(* IEC 61131-3 sources: FIOWrap/src/Ar/FIOWrap, 8 files *)

(* ---- FIOWrap.typ ---- *)
(*
 * File: FIOWrap.typ
 * Copyright (c) 2023 Loupe
 * https://loupe.team
 *
 * This file is part of FIOWrap, licensed under the MIT License.
 *
 ********************************************************************
 * Data types of library FIOWrap
 ********************************************************************)

TYPE
	FIOWRAP_ERR_enum :
		(
		FIOWRAP_ERR_INVALIDOP := 50000,
		FIOWRAP_ERR_INVALIDFILTER,
		FIOWRAP_ERR_INVALIDDIR,
		FIOWRAP_ERR_MAXFILESIZE
		);
	FIOWRAP_OP_enum :
		(
		FIOWRAP_OP_INVALID := 0,
		FIOWRAP_OP_OPEN,
		FIOWRAP_OP_SAVEAS,
		FIOWRAP_OP_APPEND,
		FIOWRAP_OP_APPEND_NEW,
		FIOWRAP_OP_SCAN,
		FIOWRAP_OP_DELETE,
		FIOWRAP_OP_DELETE_ALL,
		FIOWRAP_OP_ERROR
		);
	FIOWRAP_ST_enum :
		(
		FIOWRAP_ST_WAIT := 0, (*0*)
		FIOWRAP_ST_OPEN, (*1*)
		FIOWRAP_ST_CREATE, (*2*)
		FIOWRAP_ST_WRITE_HEADER, (*3*)
		FIOWRAP_ST_READ, (*4*)
		FIOWRAP_ST_WRITE, (*5*)
		FIOWRAP_ST_CLOSE, (*6*)
		FIOWRAP_ST_DELETE, (*7*)
		FIOWRAP_ST_DELETE_FILE, (*8*)
		FIOWRAP_ST_DELETE_DIR, (*9*)
		FIOWRAP_ST_RENAME, (*10*)
		FIOWRAP_ST_INFO, (*11*)
		FIOWRAP_ST_ERROR := 999, (*999*)
		FIOWRAP_ST_
		);
	FIOWrap_Int_FUB_typ : 	STRUCT
		Open : FileOpen;
		Create : FileCreate;
		Read : FileRead;
		Write : FileWrite;
		Close : FileClose;
		Delete : FileDelete;
		Rename : FileRename;
		GetTime : DTGetTime;
		Info : FileInfo;
	END_STRUCT;
	FIOWrap_Internal_typ : 	STRUCT
		FileID : UDINT; (*File Ident for reading and writing*)
		FileLen : UDINT; (*Length of the current file for appending*)
		FileCreated : BOOL; (*Error happened after opening file.  Need to close and then go to error state.*)
		ErrorClose : BOOL; (*Error happened after opening file.  Need to close and then go to error state.*)
		CurrOperation : DINT;
		State : DINT;
		Timestamp : STRING[30];
		newFileName : STRING[FIOWRAP_STRLEN_NAME];
		Name : STRING[FIOWRAP_STRLEN_NAME];
		Extension : STRING[FIOWRAP_STRLEN_NAME];
		FUB : FIOWrap_Int_FUB_typ;
		CMD : FIOWrap_IN_CMD_typ;
		DTStruct : DTStructure;
		TempStr : STRING[FIOWRAP_STRLEN_NAME];
		FileInfo : fiFILE_INFO;
		headerLen : UDINT;
	END_STRUCT;
	FIOWrap_OUT_STAT_typ : 	STRUCT
		Busy : BOOL;
		Done : BOOL;
		Error : BOOL;
		ErrorID : UINT;
		ErrorString : STRING[FIOWRAP_STRLEN_ERROR];
		ErrorLevel : USINT;
		ReadyForCMD : BOOL;
		NewFile : BOOL; (*Length of the current file for appending*)
		FileLen : UDINT; (*Length of the current file for appending*)
	END_STRUCT;
	FIOWrap_OUT_typ : 	STRUCT
		STAT : FIOWrap_OUT_STAT_typ;
	END_STRUCT;
	FIOWrap_IN_PAR_typ : 	STRUCT
		FileDevice : STRING[FIOWRAP_STRLEN_NAME]; (*File device name*)
		FileName : STRING[FIOWRAP_STRLEN_NAME]; (*File name (with extension)*)
		Suffix : STRING[FIOWRAP_STRLEN_NAME]; (*File name (with extension)*)
		pData : UDINT; (*Address of the data to be read or written*)
		len : UDINT; (*Length of the data to be read or written*)
		offset : UDINT; (*Offset within the file to read/write from/to.*)
		MaxFileSize : UDINT; (*Maximum file size (only evaluated when appending to a file)*)
		MultiFile : BOOL; (*Allow multiple files to be created. When true, AppendToFile will not issue an error if the MaxFileSize would be exceeded. Instead, a new file is created with the name FileName. The original file is renamed to include the FileName and the Suffix.*)
		pHeader : UDINT; (*Address of data to be added to the top of new files*)
		headerLen : UDINT; (*Length or size of header in bytes*)
	END_STRUCT;
	FIOWrap_IN_CMD_typ : 	STRUCT
		Open : BOOL; (*Open a file and read its contents*)
		SaveAs : BOOL; (*Save data to a file*)
		AppendToFile : BOOL; (*Append data to the end of a file*)
		Delete : BOOL;
		AcknowledgeError : BOOL;
	END_STRUCT;
	FIOWrap_IN_typ : 	STRUCT
		CMD : FIOWrap_IN_CMD_typ;
		PAR : FIOWrap_IN_PAR_typ;
	END_STRUCT;
	FIOWrap_typ : 	STRUCT
		IN : FIOWrap_IN_typ;
		OUT : FIOWrap_OUT_typ;
		Internal : FIOWrap_Internal_typ;
	END_STRUCT;
	FIOManage_Int_FUB_typ : 	STRUCT
		DirOpen : DirOpen;
		DirClose : DirClose;
		DirRead : DirReadEx;
		DeleteDir : DirDeleteEx;
		Delete : FileDelete;
	END_STRUCT;
	FIOManage_Internal_typ : 	STRUCT
		DirID : UDINT; (*File Ident for reading and writing*)
		NumDirs : UDINT; (*Length of the current file for appending*)
		NumItems : UDINT; (*Length of the current file for appending*)
		CurrOperation : FIOWRAP_OP_enum;
		ErrorClose : BOOL; (*Error happened after opening file.  Need to close and then go to error state.*)
		State : DINT;
		index : USINT;
		FilterName : STRING[FIOWRAP_STRLEN_NAME];
		ItemName : STRING[FIOWRAP_STRLEN_NAME];
		FileExtension : STRING[FIOWRAP_STRLEN_NAME];
		Name : STRING[FIOWRAP_STRLEN_NAME];
		Extension : STRING[FIOWRAP_STRLEN_NAME];
		NumItemsDelete : DINT;
		ItemInfo : fiDIR_READ_EX_DATA;
		ItemInfoCache : ARRAY[0..FIOWRAP_MAI_DELETE]OF fiDIR_READ_EX_DATA;
		NewestIndex : USINT;
		OldestIndex : USINT;
		FUB : FIOManage_Int_FUB_typ;
		CMD : FIOManage_IN_CMD_typ;
	END_STRUCT;
	FIOManage_OUT_STAT_typ : 	STRUCT
		Busy : BOOL;
		Done : BOOL;
		Error : BOOL;
		ErrorID : UINT;
		ErrorString : STRING[FIOWRAP_STRLEN_ERROR];
		ErrorLevel : USINT;
		ReadyForCMD : BOOL;
	END_STRUCT;
	FIOManage_OUT_typ : 	STRUCT
		STAT : FIOManage_OUT_STAT_typ;
	END_STRUCT;
	FIOManage_IN_PAR_typ : 	STRUCT
		FileDevice : STRING[FIOWRAP_STRLEN_NAME]; (*File device name*)
		Directory : STRING[FIOWRAP_STRLEN_NAME]; (*Directory to navigate to*)
		ItemName : STRING[FIOWRAP_STRLEN_NAME]; (*Address of the data to be read or written*)
		MaxNumItems : UDINT; (*Maximum file size (only evaluated when appending to a file)*)
		Mode : USINT; (*Maximum file size (only evaluated when appending to a file)*)
	END_STRUCT;
	FIOManage_IN_CMD_typ : 	STRUCT
		Scan : BOOL;
		DeleteAll : BOOL;
		AcknowledgeError : BOOL;
	END_STRUCT;
	FIOManage_IN_typ : 	STRUCT
		CMD : FIOManage_IN_CMD_typ;
		PAR : FIOManage_IN_PAR_typ;
	END_STRUCT;
	FIOManage_typ : 	STRUCT
		IN : FIOManage_IN_typ;
		OUT : FIOManage_OUT_typ;
		Internal : FIOManage_Internal_typ;
	END_STRUCT;
END_TYPE

(* ---- FIOManageFn_Cyclic.st ---- *)
(*
 * File: FIOManageFn_Cyclic.st
 * Copyright (c) 2023 Loupe
 * https://loupe.team
 *
 * This file is part of FIOWrap, licensed under the MIT License.
 *
  ********************************************************************
 * Implementation of library FIOWrap
 ********************************************************************)

(********************************************************************)
(* This function manages multiple files for logs					*)
(********************************************************************)

(* Resetting internal CMDs				DONE and NOT TESTED *)

(* Main State machine					DONE NOT TESTED *)

	(* ST_WAIT							DONE NOT TESTED *)
		(* Wait for new CMDs			DONE and TESTED *)
			(* Scan						DONE and TESTED  *)
				(* Set CurrOperation	DONE and TESTED  *)
				(* Busy, Done			DONE and TESTED  *)
				(* Change state			DONE and TESTED  *)
			(* DeleteAll				DONE and NOT TESTED  *)
				(* Set CurrOperation	DONE and TESTED  *)
				(* Busy, Done			DONE and TESTED  *)
				(* Change state			DONE and TESTED  *)
		(* Reset Done					DONE and TESTED  *)

	(* ST_OPEN							DONE and NOT TESTED  *)
		(* FUB inputs					DONE and TESTED  *)
		(* Status checking				DONE and TESTED  *)
			(* Done						DONE and TESTED  *)
			(* No error					DONE and TESTED  *)
				(* Open					DONE and TESTED  *)
			(* Other error				DONE and NOT TESTED  *)

	(* ST_READ							DONE and NOT TESTED  *)
		(* FUB inputs					DONE and NOT TESTED  *)
		(* Status checking				DONE and NOT TESTED  *)
			(* Done						DONE and TESTED  *)
			(* No error					DONE and TESTED  *)
			(* Error					DONE and TESTED  *)

	(* ST_CLOSE							DONE and NOT TESTED  *)
		(* FUB inputs					DONE and NOT TESTED  *)
		(* Status checking				DONE and NOT TESTED  *)
			(* Done						DONE and TESTED  *)
			(* No error					DONE and TESTED  *)
				(* ErrorClose			DONE and NOT TESTED  *)
			(* Error					DONE will not be tested *)

	(* ST_DELETE						DONE and NOT TESTED  *)
		(* FUB inputs					DONE and NOT TESTED  *)
		(* Status checking				DONE and NOT TESTED  *)
			(* Done						DONE and TESTED  *)
			(* No error					DONE and TESTED  *)
			(* File not found			DONE and NOT TESTED  *)
			(* Other error				DONE and NOT TESTED  *)

	(* ST_ERROR							DONE and TESTED  *)
		(* Disable FUBs					DONE and TESTED  *)
		(* AcknowledgeError CMD			DONE and TESTED  *)

(* Busy, Done, Error					DONE and TESTED  *)

FUNCTION FIOManageFn_Cyclic

(************************************************************************)
(* Set return value to get rid of compiler warning 						*)
(************************************************************************)

FIOManageFn_Cyclic:=	FALSE;

(************************************************************************)
(* Reset internal CMDs													*)
(************************************************************************)

IF( NOT(t.IN.CMD.Scan) )THEN

	t.Internal.CMD.Scan:=	0;

END_IF

IF( NOT(t.IN.CMD.DeleteAll) )THEN

	t.Internal.CMD.DeleteAll:=	0;

END_IF

(************************************************************************)
(* Main state machine													*)
(************************************************************************)

	CASE t.Internal.State OF

		FIOWRAP_ST_WAIT:

			(* If all CMDs are cleared, then clear Done status *)

			IF( 	NOT(t.IN.CMD.Scan)
				AND	NOT(t.IN.CMD.DeleteAll)
				)THEN

				t.OUT.STAT.Done:=	0;

			END_IF

			(* Set CurrOperation to INVALID. It will be set below on leaving the state *)

			t.Internal.CurrOperation:=	FIOWRAP_OP_INVALID;

			(* Wait for new commands *)

			IF( t.IN.CMD.Scan AND NOT(t.Internal.CMD.Scan) )THEN

				t.Internal.CMD.Scan:=	1;

				t.OUT.STAT.Busy:=	1;
				t.OUT.STAT.Done:=	0;

				t.Internal.State:=			FIOWRAP_ST_OPEN;
				t.Internal.CurrOperation:=	FIOWRAP_OP_SCAN;

				// Modify filter based off of input itemName
				IF(t.IN.PAR.ItemName = '') THEN
					// Set error for filter input
					fiomSetError( DINT_TO_UINT(FIOWRAP_ERR_INVALIDFILTER), t );
				ELSIF (t.IN.PAR.ItemName = '*') THEN
					t.Internal.FilterName := '';
				ELSE
					t.Internal.FilterName := t.IN.PAR.ItemName;
				END_IF

			ELSIF( t.IN.CMD.DeleteAll AND NOT(t.Internal.CMD.DeleteAll) )THEN

				// TODO: Delete All should not open file more than once

				t.Internal.CMD.DeleteAll:=	1;

				t.OUT.STAT.Busy:=	1;
				t.OUT.STAT.Done:=	0;

				t.Internal.State:=			FIOWRAP_ST_OPEN;
				t.Internal.CurrOperation:=	FIOWRAP_OP_DELETE_ALL;

			END_IF

		FIOWRAP_ST_OPEN:

			(* Open Dir *)

			t.Internal.FUB.DirOpen.enable:=	1;
			t.Internal.FUB.DirOpen.pDevice:=	ADR(t.IN.PAR.FileDevice);
			IF( brsstrlen(ADR(t.IN.PAR.Directory)) = 0 )THEN
				t.Internal.FUB.DirOpen.pName:= 0;
				// Scanning/deleting is not allowed while in a root directory
				// TODO: figure out how to throw an error because figuring out if you are in a root directory is difficult
			ELSE
				t.Internal.FUB.DirOpen.pName:=		ADR(t.IN.PAR.Directory);
			END_IF

			(* Check status *)

			IF( t.Internal.FUB.DirOpen.status < FIOWRAP_STAT_DISABLED ) THEN

				(* Turn off FUB *)

				t.Internal.FUB.DirOpen.enable:=	0;

				IF( t.Internal.FUB.DirOpen.status = FIOWRAP_STAT_OK ) THEN

				(* All good
					Get Ident, go to appropriate state *)

					t.Internal.DirID:=		t.Internal.FUB.DirOpen.ident;

					IF( t.Internal.CurrOperation = FIOWRAP_OP_DELETE
						OR t.Internal.CurrOperation = FIOWRAP_OP_DELETE_ALL
						OR t.Internal.CurrOperation = FIOWRAP_OP_SCAN)THEN

						t.Internal.State:= FIOWRAP_ST_READ;

					ELSE

						fiomSetError( DINT_TO_UINT(FIOWRAP_ERR_INVALIDOP), t );

					END_IF

				ELSE

					(* Other error *)

					fiomSetError( t.Internal.FUB.DirOpen.status, t );

				END_IF (* If error *)

		END_IF (* If done *)

		FIOWRAP_ST_READ:

			(* Check status *)

			IF( t.Internal.FUB.DirRead.status < FIOWRAP_STAT_DISABLED )THEN

				(* Turn off FUB *)

				t.Internal.FUB.DirRead.enable:= 0;

				IF ( t.Internal.FUB.DirRead.status = FIOWRAP_STAT_OK ) THEN

					(* Turn on FUB *)
					t.Internal.FUB.DirRead.enable:= 1;

					// Check mode and file type before adding to the cache
					IF( (t.IN.PAR.Mode = fiFILE AND t.Internal.ItemInfo.Mode = fiFILE)
						OR (t.IN.PAR.Mode = fiDIRECTORY AND t.Internal.ItemInfo.Mode = fiDIRECTORY)
						OR (t.IN.PAR.Mode = fiBOTH) )THEN

						(* Get File Names and Extensions *)
						SplitFileName(ADR(t.Internal.FilterName),ADR(t.Internal.Name), ADR(t.Internal.Extension));
						SplitFileName(ADR(t.Internal.ItemInfo.Filename),0,ADR(t.Internal.FileExtension));
						brsmemcpy(ADR(t.Internal.ItemName),ADR(t.Internal.ItemInfo.Filename),brsstrlen(ADR(t.Internal.Name)));

						// Check to see if the file/directory name and extension (if specified) match and that the directory is not '.' or '..'
						IF( (brsstrcmp(ADR(t.Internal.ItemName),ADR(t.Internal.Name)) = 0)
							AND ((brsstrcmp(ADR(t.Internal.FileExtension),ADR(t.Internal.Extension)) = 0) OR (brsstrcmp(ADR(t.Internal.Extension),ADR('')) = 0))
							AND NOT ((brsstrcmp(ADR(t.Internal.ItemInfo.Filename),ADR('.')) = 0) OR (brsstrcmp(ADR(t.Internal.ItemInfo.Filename),ADR('..')) = 0) ))THEN
							// increment number of files
							t.Internal.NumItems:= t.Internal.NumItems+1;

							// All indices in the cache are set to very large dates initially
							IF( t.Internal.ItemInfoCache[t.Internal.NewestIndex].Date > t.Internal.ItemInfo.Date )THEN

								(* Record Older file info *)
								brsmemcpy(ADR(t.Internal.ItemInfoCache[t.Internal.NewestIndex]),ADR(t.Internal.ItemInfo),SIZEOF(t.Internal.ItemInfo));

								(* Find Oldest / Newest file *)
								FOR t.Internal.index := 0 TO FIOWRAP_MAI_DELETE DO
									IF t.Internal.ItemInfoCache[t.Internal.OldestIndex].Date > t.Internal.ItemInfoCache[t.Internal.index].Date THEN
										t.Internal.OldestIndex := t.Internal.index;
									END_IF
									IF  t.Internal.ItemInfoCache[t.Internal.NewestIndex].Date < t.Internal.ItemInfoCache[t.Internal.index].Date THEN
										t.Internal.NewestIndex := t.Internal.index;
									END_IF
								END_FOR;
							END_IF

							// Start deleting files if you have the max number of files you can delete in one read.
							IF( t.Internal.NumItems >=  FIOWRAP_NUM_DELETE
								AND t.Internal.CurrOperation = FIOWRAP_OP_DELETE_ALL )THEN

								t.Internal.FUB.DirRead.enable:= 0;

								t.Internal.NumItemsDelete:= FIOWRAP_NUM_DELETE;

								(* Delete files *)

								t.Internal.State := FIOWRAP_ST_DELETE;

							END_IF

						END_IF

					END_IF

				ELSIF ( t.Internal.FUB.DirRead.status = fiERR_NO_MORE_ENTRIES ) THEN

					IF t.Internal.CurrOperation = FIOWRAP_OP_DELETE_ALL THEN

						(* Delete Files *)

						t.Internal.NumItemsDelete:= MIN(t.Internal.NumItems, FIOWRAP_NUM_DELETE);

						IF t.Internal.NumItemsDelete > 0 THEN
							t.Internal.CurrOperation := FIOWRAP_OP_DELETE;
						ELSE
							t.Internal.CurrOperation := FIOWRAP_OP_SCAN; //TODO: Change this to valid op
						END_IF

					ELSIF t.Internal.NumItems > t.IN.PAR.MaxNumItems THEN

						(* Delete Files *)

						t.Internal.NumItemsDelete:= MIN(t.Internal.NumItems - t.IN.PAR.MaxNumItems, FIOWRAP_NUM_DELETE);

						t.Internal.CurrOperation := FIOWRAP_OP_DELETE;

					END_IF

					IF( t.Internal.CurrOperation = FIOWRAP_OP_DELETE
						OR t.Internal.CurrOperation = FIOWRAP_OP_DELETE_ALL
						OR t.Internal.CurrOperation = FIOWRAP_OP_SCAN )THEN

						(* Close Dir *)

						t.Internal.State := FIOWRAP_ST_CLOSE;

					ELSE

						fiomSetError( DINT_TO_UINT(FIOWRAP_ERR_INVALIDOP), t );

					END_IF

				ELSE

					(* Error *)

					t.Internal.ErrorClose:= 1;

					IF( t.Internal.FUB.DirRead.status = 20799 )THEN

						//If the sysError ID = 65535 then we are in a root directory and can't do a read
						t.OUT.STAT.ErrorID := FileIoGetSysError();
						IF (t.OUT.STAT.ErrorID = 65535) THEN
							fiomSetError( DINT_TO_UINT(FIOWRAP_ERR_INVALIDDIR), t );
						ELSE
							fiomSetError( t.OUT.STAT.ErrorID, t );
						END_IF

					ELSE

						fiomSetError( t.Internal.FUB.DirRead.status, t );

					END_IF

					t.Internal.State:= FIOWRAP_ST_CLOSE;

				END_IF

			ELSIF( t.Internal.FUB.DirRead.status = FIOWRAP_STAT_DISABLED )THEN

				(* Enable FUB *)
				t.Internal.FUB.DirRead.enable 	:= 1;
				t.Internal.FUB.DirRead.ident	:= t.Internal.DirID;
				t.Internal.FUB.DirRead.pData	:= ADR(t.Internal.ItemInfo);
				t.Internal.FUB.DirRead.data_len	:= SIZEOF(t.Internal.ItemInfo);

				t.Internal.NumItems := 0;
				t.Internal.NumItemsDelete:= 0;
				t.Internal.OldestIndex := 0;
				t.Internal.NewestIndex := 0;
				brsmemset(ADR(t.Internal.ItemName), 0, SIZEOF(t.Internal.ItemName));

				brsmemset(ADR(t.Internal.ItemInfoCache), 0, SIZEOF(t.Internal.ItemInfoCache));
				FOR t.Internal.index := 0 TO FIOWRAP_MAI_DELETE DO
					t.Internal.ItemInfoCache[t.Internal.index].Date := DT#2106-02-06-06:28:15; // Can this be a hex value instead?
				END_FOR

			END_IF

		FIOWRAP_ST_CLOSE:

			(* Close file *)

			t.Internal.FUB.DirClose.enable:=	1;
			t.Internal.FUB.DirClose.ident:=	t.Internal.DirID;

			(* Check status *)

			IF( t.Internal.FUB.DirClose.status < FIOWRAP_STAT_DISABLED ) THEN

				(* Turn off FUB *)

				t.Internal.FUB.DirClose.enable:=	0;

				IF( t.Internal.FUB.DirClose.status = FIOWRAP_STAT_OK ) THEN

					IF( t.Internal.ErrorClose ) THEN

						(* If error, go to error state *)

						t.Internal.State:=	FIOWRAP_ST_ERROR;

						t.Internal.ErrorClose:= 0;

					ELSIF( (t.Internal.CurrOperation = FIOWRAP_OP_DELETE
						OR t.Internal.CurrOperation = FIOWRAP_OP_DELETE_ALL)
						AND t.Internal.NumItemsDelete > 0) THEN

						t.Internal.State:=	FIOWRAP_ST_DELETE;

					ELSE

						(* otherwise, done, set status and go to wait state *)

						t.OUT.STAT.Busy:=	0;
						t.OUT.STAT.Done:=	1;

						t.Internal.State:=	FIOWRAP_ST_WAIT;

					END_IF (* If ErrorClose *)

				ELSE

					(* Error *)

					fiomSetError( t.Internal.FUB.DirClose.status, t );

				END_IF (* If error *)

		END_IF (*If done *)

		FIOWRAP_ST_DELETE:

			IF( t.Internal.NumItemsDelete > 0 )THEN

				(* Generate file name *)

				brsmemcpy(ADR(t.Internal.ItemName),ADR(t.Internal.ItemInfoCache[t.Internal.OldestIndex].Filename),SIZEOF(t.Internal.ItemName));
				t.Internal.ItemName := CONCAT(CONCAT(t.IN.PAR.Directory, '/'), t.Internal.ItemName);

				// Check file type and go to appropriate state
				IF(t.Internal.ItemInfoCache[t.Internal.OldestIndex].Mode = fiFILE) THEN
					t.Internal.State := FIOWRAP_ST_DELETE_FILE;
				ELSE
					t.Internal.State := FIOWRAP_ST_DELETE_DIR;
				END_IF

				(* Remove Old file from list *)

				t.Internal.ItemInfoCache[t.Internal.OldestIndex].Date := DT#2106-02-06-06:28:15; // Can this be a hex value instead?

				(* Find new oldest / newest file *)

				FOR t.Internal.index := 0 TO FIOWRAP_MAI_DELETE DO
					IF t.Internal.ItemInfoCache[t.Internal.OldestIndex].Date > t.Internal.ItemInfoCache[t.Internal.index].Date THEN
						t.Internal.OldestIndex := t.Internal.index;
					END_IF
					IF  t.Internal.ItemInfoCache[t.Internal.NewestIndex].Date < t.Internal.ItemInfoCache[t.Internal.index].Date THEN
						t.Internal.NewestIndex := t.Internal.index;
					END_IF
				END_FOR;

			ELSIF( t.Internal.NumItemsDelete <= 0 )THEN

				IF( t.Internal.CurrOperation = FIOWRAP_OP_DELETE_ALL )THEN

					(* Go to Read *)
					// Find more files to delete
					t.Internal.State:= FIOWRAP_ST_OPEN;

				ELSIF( t.Internal.CurrOperation = FIOWRAP_OP_DELETE )THEN

					(* Done, set status and go to wait state *)
					t.OUT.STAT.Busy:=	0;
					t.OUT.STAT.Done:=	1;

					t.Internal.State:=	FIOWRAP_ST_WAIT;

				ELSE
					// Set the error
					fiomSetError( DINT_TO_UINT(FIOWRAP_ERR_INVALIDOP), t );

				END_IF

			END_IF

		FIOWRAP_ST_DELETE_FILE:
			(* Enable FUB *)
			IF (NOT t.Internal.FUB.Delete.enable) THEN
				t.Internal.FUB.Delete.enable := 1;
				t.Internal.FUB.Delete.pDevice := ADR(t.IN.PAR.FileDevice);
				t.Internal.FUB.Delete.pName := ADR(t.Internal.ItemName);
			END_IF

			(*Delete File*)
			IF( t.Internal.FUB.Delete.status < FIOWRAP_STAT_DISABLED )THEN

				(* Turn off FUB *)
				t.Internal.FUB.Delete.enable:= 0;

				IF( t.Internal.FUB.Delete.status = FIOWRAP_STAT_OK )THEN

					t.Internal.NumItems := t.Internal.NumItems - 1;
					t.Internal.NumItemsDelete := t.Internal.NumItemsDelete - 1;

					// Return to delete state
					t.Internal.State := FIOWRAP_ST_DELETE;

				ELSE

					(* error *)

					//TODO: Handle file not found error

					fiomSetError( t.Internal.FUB.Delete.status, t );

				END_IF
			END_IF

		FIOWRAP_ST_DELETE_DIR:
			(* Enable FUB *)
			IF (NOT t.Internal.FUB.DeleteDir.enable) THEN
				t.Internal.FUB.DeleteDir.enable := 1;
				t.Internal.FUB.DeleteDir.pDevice := ADR(t.IN.PAR.FileDevice);
				t.Internal.FUB.DeleteDir.pName := ADR(t.Internal.ItemName);
			END_IF

			(*Delete File*)

			IF( t.Internal.FUB.DeleteDir.status < FIOWRAP_STAT_DISABLED )THEN

				(* Turn off FUB *)

				t.Internal.FUB.DeleteDir.enable:= 0;

				IF( t.Internal.FUB.DeleteDir.status = FIOWRAP_STAT_OK )THEN

					t.Internal.NumItems := t.Internal.NumItems - 1;
					t.Internal.NumItemsDelete := t.Internal.NumItemsDelete - 1;

					// Return to delete state
					t.Internal.State := FIOWRAP_ST_DELETE;

				ELSE

					(* error *)

					//TODO: Handle file not found error

					fiomSetError( t.Internal.FUB.DeleteDir.status, t );

				END_IF
			END_IF

		FIOWRAP_ST_ERROR:

			(* Turn off all FUBs, just in case *)

			t.Internal.FUB.DirOpen.enable:=	0;
			t.Internal.FUB.DirRead.enable:=	0;
			t.Internal.FUB.DirClose.enable:=	0;
			t.Internal.FUB.Delete.enable:=	0;

			IF( t.IN.CMD.AcknowledgeError )THEN

				t.OUT.STAT.Error:=			0;
				t.OUT.STAT.ErrorID:=		0;
				t.OUT.STAT.ErrorString:=	'';
				t.OUT.STAT.ErrorLevel:=		0;
				t.Internal.State:=			FIOWRAP_ST_WAIT;

			END_IF

	END_CASE

	(* Reset AcknowledgeError CMD *)

	t.IN.CMD.AcknowledgeError:=	0;

	(****************************************)
	(* Call FUBs							*)
	(****************************************)

	t.Internal.FUB.DirOpen();
	t.Internal.FUB.DirRead();
	t.Internal.FUB.DirClose();
	t.Internal.FUB.Delete();
	t.Internal.FUB.DeleteDir();

(****************************************)
(* Set ReadyForCMD						*)
(****************************************)

t.OUT.STAT.ReadyForCMD:=		NOT(t.OUT.STAT.Busy)
							AND NOT(t.OUT.STAT.Done)
							AND	NOT(t.OUT.STAT.Error);

END_FUNCTION

(* ---- fiomSetError.st ---- *)
(*
 * File: fiomSetError.st
 * Copyright (c) 2023 Loupe
 * https://loupe.team
 *
 * This file is part of FIOWrap, licensed under the MIT License.
 *
  ********************************************************************
 * Implementation of library FIOWrap
 ********************************************************************)

(********************************************************************)
(* Set error status on FIOWrap 										*)
(********************************************************************)

(* Reset Busy, Done			DONE and TESTED DFB 20111222 *)
(* Set Error				DONE and TESTED DFB 20111222 *)
(* Set ErrorID				DONE and TESTED DFB 20111222 *)
(* Set ErrorLevel			DONE and TESTED DFB 20111222 *)
(* Set State				DONE and TESTED DFB 20111222 *)
(* Set ErrorString			DONE and TESTED DFB 20120131 *)

FUNCTION fiomSetError

(****************************************************)
(* Set return value to get rid of compile warning 	*)
(****************************************************)

fiomSetError:=	FALSE;

(************************************************)
(* Set error status								*)
(************************************************)

t.OUT.STAT.Busy:=		0;
t.OUT.STAT.Done:=		0;
t.OUT.STAT.Error:=		1;
t.OUT.STAT.ErrorID:=	ErrorID;
t.OUT.STAT.ErrorLevel:=	3;
t.Internal.State:=		FIOWRAP_ST_ERROR;

(* Set ErrorString *)

CASE ErrorID OF

	0: t.OUT.STAT.ErrorString:=	'';

	fiERR_INVALID_PATH:				t.OUT.STAT.ErrorString:=	'Invalid path.';
	fiERR_DATA_SIZE:				t.OUT.STAT.ErrorString:=	'Data length is too small (DirRead).';
	fiERR_NO_MORE_ENTRIES:			t.OUT.STAT.ErrorString:=	'No more file handles available.';
	fiERR_NOT_SUPPORTED:			t.OUT.STAT.ErrorString:=	'System error.';
	fiERR_INVALID_TYP:				t.OUT.STAT.ErrorString:=	'Invalid type.';
	fiERR_EXIST:					t.OUT.STAT.ErrorString:=	'File already exists.';
	fiERR_ACCESS:					t.OUT.STAT.ErrorString:=	'Access not possible with the desired mode.';
	fiERR_MODE:						t.OUT.STAT.ErrorString:=	'Illegal mode.';
	fiERR_FILE_NOT_FOUND:			t.OUT.STAT.ErrorString:=	'File not found. Check IN.PAR.FileName.';
	fiERR_FILE_DEVICE:				t.OUT.STAT.ErrorString:=	'File device not found. Check IN.PAR.FileDevice.';
	fiERR_SPACE:					t.OUT.STAT.ErrorString:=	'Not enough memory to write file.';
	fiERR_SEEK:						t.OUT.STAT.ErrorString:=	'Invalid file offset.';
	fiERR_FILE:						t.OUT.STAT.ErrorString:=	'File not allowed.';
	fiERR_LESS_VIRTUAL_MEMORY:		t.OUT.STAT.ErrorString:=	'Not enough memory to write file.';
	fiERR_COM_FILE_OPEN:			t.OUT.STAT.ErrorString:=	'System error.';
	fiERR_COM_FILE_CLOSE:			t.OUT.STAT.ErrorString:=	'System error.';
	fiERR_COM_FILE_READ:			t.OUT.STAT.ErrorString:=	'System error.';
	fiERR_COM_FILE_WRITE:			t.OUT.STAT.ErrorString:=	'System error.';
	fiERR_COM_FILE_IOCTL:			t.OUT.STAT.ErrorString:=	'System error.';
	fiERR_DATA:						t.OUT.STAT.ErrorString:=	'Invalid parameter. Check IN.PAR.pData.';
	fiERR_ASYNC_MANAGER:			t.OUT.STAT.ErrorString:=	'System error.';
	fiERR_FILE_NOT_OPENED:			t.OUT.STAT.ErrorString:=	'File not opened.';
	fiERR_INVALID_DIRECTORY:		t.OUT.STAT.ErrorString:=	'Invalid directory. Check IN.PAR.FileDevice and IN.PAR.FileDirectory.';
	fiERR_DIR_NOT_EXIST:			t.OUT.STAT.ErrorString:=	'Directory does not exist. Check IN.PAR.FileDevice and IN.PAR.FileDirectory.';
	fiERR_DIR_NOT_EMPTY:			t.OUT.STAT.ErrorString:=	'Directory is not empty.';
	fiERR_DIR_ALREADY_EXIST:		t.OUT.STAT.ErrorString:=	'Directory already exists.';
	fiERR_DETMEMINFO:				t.OUT.STAT.ErrorString:=	'System error.';
	fiERR_NOT_ENOUGH_FREEMEM:		t.OUT.STAT.ErrorString:=	'Not enough memory to write file.';
	fiERR_DIR_INVALID_HANDLE:		t.OUT.STAT.ErrorString:=	'System error.';
	fiERR_PARAMETER:				t.OUT.STAT.ErrorString:=	'System error.';
	fiERR_DEVICE_ALREADY_EXIST:		t.OUT.STAT.ErrorString:=	'Device already exists.';
	fiERR_DEVICE_INVALID_HANDLE:	t.OUT.STAT.ErrorString:=	'Invalid device handle.';
	fiERR_NETIO_IP_UNEQUAL:			t.OUT.STAT.ErrorString:=	'IP address error. Check hostname.';
	fiERR_INIT:						t.OUT.STAT.ErrorString:=	'System error.';
	fiERR_DEVICE_DRIVER:			t.OUT.STAT.ErrorString:=	'System error.';
	fiERR_DEVICE_MANAGER:			t.OUT.STAT.ErrorString:=	'File device error. Check IN.PAR.FileDevice.';
	fiERR_SYSTEM:					t.OUT.STAT.ErrorString:=	'System error.';

	FIOWRAP_ERR_INVALIDOP:			t.OUT.STAT.ErrorString:=	'Internal error.';
	FIOWRAP_ERR_INVALIDFILTER:		t.OUT.STAT.ErrorString:=	'Input required for IN.PAR.ItemName. Set IN.PAR.ItemName := $'*$' to mamange all files/directories.';
	FIOWRAP_ERR_INVALIDDIR:			t.OUT.STAT.ErrorString:=	'Cannot manage in root directory. Check IN.PAR.FileDevice and IN.PAR.FileDirectory.';
	FIOWRAP_ERR_MAXFILESIZE:		t.OUT.STAT.ErrorString:=	'Error while appending: maximum file size would be exceeded.';

	ELSE	t.OUT.STAT.ErrorString:=	'Unknown error.';

END_CASE

END_FUNCTION

(* ---- fioOpenFile_Init.st ---- *)
(*
 * File: fioOpenFile_Init.st
 * Copyright (c) 2023 Loupe
 * https://loupe.team
 *
 * This file is part of FIOWrap, licensed under the MIT License.
 *
 *)

//-------------------------------------------------------------------
// Open a file in the init subroutine
//-------------------------------------------------------------------

FUNCTION fioOpenFile_Init

	// Open a file - tested
	WHILE (TRUE) DO

		t.IN.CMD.Open := TRUE;

		FIOWrapFn_Cyclic(t);

		IF (t.OUT.STAT.Done OR t.OUT.STAT.Error) THEN
			t.IN.CMD.Open := FALSE;
			FIOWrapFn_Cyclic(t);
			fioOpenFile_Init := t.OUT.STAT.ErrorID;
			RETURN;
		END_IF

	END_WHILE

END_FUNCTION

(* ---- FIOWrap.fun ---- *)
(*
 * File: FIOWrap.fun
 * Copyright (c) 2023 Loupe
 * https://loupe.team
 *
 * This file is part of FIOWrap, licensed under the MIT License.
 *
 ********************************************************************
 * Functions and function blocks of library FIOWrap
 ********************************************************************)

FUNCTION FIOManageFn_Cyclic : BOOL
	VAR_IN_OUT
		t : FIOManage_typ;
	END_VAR
END_FUNCTION

FUNCTION FIOWrapFn_Cyclic : BOOL (*This function manages file reads and writes.*)
	VAR_IN_OUT
		t : FIOWrap_typ; (*FIOWrap Mgr structure*)
	END_VAR
END_FUNCTION

FUNCTION fiowSetError : BOOL (*Set error status on FIOWrap*)
	VAR_INPUT
		ErrorID : UINT;
	END_VAR
	VAR_IN_OUT
		t : FIOWrap_typ;
	END_VAR
END_FUNCTION

FUNCTION fiomSetError : BOOL
	VAR_INPUT
		ErrorID : UINT;
	END_VAR
	VAR_IN_OUT
		t : FIOManage_typ;
	END_VAR
END_FUNCTION

{REDUND_ERROR} FUNCTION fioOpenFile_Init : UINT (*Open a file in the init subroutine*) (*$GROUP=User,$CAT=User,$GROUPICON=User.png,$CATICON=User.png*)
	VAR_IN_OUT
		t : FIOWrap_typ;
	END_VAR
END_FUNCTION

(* ---- fiowSetError.st ---- *)
(*
 * File: fiowSetError.st
 * Copyright (c) 2023 Loupe
 * https://loupe.team
 *
 * This file is part of FIOWrap, licensed under the MIT License.
 *
 ********************************************************************
 * Implementation of library FIOWrap
 ********************************************************************)

(********************************************************************)
(* Set error status on FIOWrap 										*)
(********************************************************************)

(* Reset Busy, Done			DONE and TESTED DFB 20111222 *)
(* Set Error				DONE and TESTED DFB 20111222 *)
(* Set ErrorID				DONE and TESTED DFB 20111222 *)
(* Set ErrorLevel			DONE and TESTED DFB 20111222 *)
(* Set State				DONE and TESTED DFB 20111222 *)
(* Set ErrorString			DONE and TESTED DFB 20120131 *)

FUNCTION fiowSetError

(****************************************************)
(* Set return value to get rid of compile warning 	*)
(****************************************************)

fiowSetError:=	FALSE;

(************************************************)
(* Set error status								*)
(************************************************)

t.OUT.STAT.Busy:=		0;
t.OUT.STAT.Done:=		0;
t.OUT.STAT.Error:=		1;
t.OUT.STAT.ErrorID:=	ErrorID;
t.OUT.STAT.ErrorLevel:=	3;
t.Internal.State:=		FIOWRAP_ST_ERROR;

(* Set ErrorString *)

CASE ErrorID OF

	0: t.OUT.STAT.ErrorString:=	'';

	fiERR_INVALID_PATH:				t.OUT.STAT.ErrorString:=	'Invalid path.';
	fiERR_DATA_SIZE:				t.OUT.STAT.ErrorString:=	'Data length is too small (DirRead).';
	fiERR_NO_MORE_ENTRIES:			t.OUT.STAT.ErrorString:=	'No more file handles available.';
	fiERR_NOT_SUPPORTED:			t.OUT.STAT.ErrorString:=	'System error.';
	fiERR_INVALID_TYP:				t.OUT.STAT.ErrorString:=	'Invalid type.';
	fiERR_EXIST:					t.OUT.STAT.ErrorString:=	'File already exists.';
	fiERR_ACCESS:					t.OUT.STAT.ErrorString:=	'Access not possible with the desired mode.';
	fiERR_MODE:						t.OUT.STAT.ErrorString:=	'Illegal mode.';
	fiERR_FILE_NOT_FOUND:			t.OUT.STAT.ErrorString:=	'File not found. Check IN.PAR.FileName.';
	fiERR_FILE_DEVICE:				t.OUT.STAT.ErrorString:=	'File device not found. Check IN.PAR.FileDevice.';
	fiERR_SPACE:					t.OUT.STAT.ErrorString:=	'Not enough memory to write file.';
	fiERR_SEEK:						t.OUT.STAT.ErrorString:=	'Invalid file offset.';
	fiERR_FILE:						t.OUT.STAT.ErrorString:=	'File not allowed.';
	fiERR_LESS_VIRTUAL_MEMORY:		t.OUT.STAT.ErrorString:=	'Not enough memory to write file.';
	fiERR_COM_FILE_OPEN:			t.OUT.STAT.ErrorString:=	'System error.';
	fiERR_COM_FILE_CLOSE:			t.OUT.STAT.ErrorString:=	'System error.';
	fiERR_COM_FILE_READ:			t.OUT.STAT.ErrorString:=	'System error.';
	fiERR_COM_FILE_WRITE:			t.OUT.STAT.ErrorString:=	'System error.';
	fiERR_COM_FILE_IOCTL:			t.OUT.STAT.ErrorString:=	'System error.';
	fiERR_DATA:						t.OUT.STAT.ErrorString:=	'Invalid parameter. Check IN.PAR.pData.';
	fiERR_ASYNC_MANAGER:			t.OUT.STAT.ErrorString:=	'System error.';
	fiERR_FILE_NOT_OPENED:			t.OUT.STAT.ErrorString:=	'File not opened.';
	fiERR_INVALID_DIRECTORY:		t.OUT.STAT.ErrorString:=	'Invalid directory. Check IN.PAR.FileDevice and IN.PAR.FileName.';
	fiERR_DIR_NOT_EXIST:			t.OUT.STAT.ErrorString:=	'Directory does not exist. Check IN.PAR.FileDevice and IN.PAR.FileName.';
	fiERR_DIR_NOT_EMPTY:			t.OUT.STAT.ErrorString:=	'Directory is not empty.';
	fiERR_DIR_ALREADY_EXIST:		t.OUT.STAT.ErrorString:=	'Directory already exists.';
	fiERR_DETMEMINFO:				t.OUT.STAT.ErrorString:=	'System error.';
	fiERR_NOT_ENOUGH_FREEMEM:		t.OUT.STAT.ErrorString:=	'Not enough memory to write file.';
	fiERR_DIR_INVALID_HANDLE:		t.OUT.STAT.ErrorString:=	'System error.';
	fiERR_PARAMETER:				t.OUT.STAT.ErrorString:=	'System error.';
	fiERR_DEVICE_ALREADY_EXIST:		t.OUT.STAT.ErrorString:=	'Device already exists.';
	fiERR_DEVICE_INVALID_HANDLE:	t.OUT.STAT.ErrorString:=	'Invalid device handle.';
	fiERR_NETIO_IP_UNEQUAL:			t.OUT.STAT.ErrorString:=	'IP address error. Check hostname.';
	fiERR_INIT:						t.OUT.STAT.ErrorString:=	'System error.';
	fiERR_DEVICE_DRIVER:			t.OUT.STAT.ErrorString:=	'System error.';
	fiERR_DEVICE_MANAGER:			t.OUT.STAT.ErrorString:=	'File device error. Check IN.PAR.FileDevice.';
	fiERR_SYSTEM:					t.OUT.STAT.ErrorString:=	'System error.';

	FIOWRAP_ERR_INVALIDOP:			t.OUT.STAT.ErrorString:=	'Internal error.';
	FIOWRAP_ERR_MAXFILESIZE:		t.OUT.STAT.ErrorString:=	'Error while appending: maximum file size would be exceeded.';

	ELSE	t.OUT.STAT.ErrorString:=	'Unknown error.';

END_CASE

END_FUNCTION

(* ---- FIOWrap.var ---- *)
(*
 * File: FIOWrap.var
 * Copyright (c) 2023 Loupe
 * https://loupe.team
 *
 * This file is part of FIOWrap, licensed under the MIT License.
 *
 ********************************************************************
 * Constants of library FIOWrap
 ********************************************************************)
VAR CONSTANT
	FIOWRAP_STRLEN_ERROR : USINT := 120;
	FIOWRAP_NUM_DELETE : USINT := 10;
	FIOWRAP_MAI_DELETE : USINT := FIOWRAP_NUM_DELETE-1;
	FIOWRAP_STRLEN_NAME : UINT := 260;
	FIOWRAP_STAT_OK : UINT := 0;
	FIOWRAP_STAT_DISABLED : UINT := 65534;
END_VAR

(* ---- FIOWrapFn_Cyclic.st ---- *)
(*
 * File: FIOWrapFn_Cyclic.st
 * Copyright (c) 2023 Loupe
 * https://loupe.team
 *
 * This file is part of FIOWrap, licensed under the MIT License.
 *
 ********************************************************************
 * Implementation of library FIOWrap
 ********************************************************************)

(********************************************************************)
(* This function manages simple file reads and writes				*)
(********************************************************************)

(* Resetting internal CMDs				DONE and TESTED DFB 20110602 *)

(* Main State machine					DONE and TESTED DFB 20110602 *)

	(* ST_WAIT							DONE and TESTED DFB 20110602 *)
		(* Wait for new CMDs			DONE and TESTED DFB 20110602 *)
			(* SaveAs					DONE and TESTED DFB 20110602 *)
				(* Set CurrOperation	DONE and TESTED DFB 20110602 *)
				(* Busy, Done			DONE and TESTED DFB 20110602 *)
				(* Change state			DONE and TESTED DFB 20110602 *)
			(* Open						DONE and TESTED DFB 20110602 *)
				(* Set CurrOperation	DONE and TESTED DFB 20110602 *)
				(* Busy, Done			DONE and TESTED DFB 20110602 *)
				(* Change state			DONE and TESTED DFB 20110602 *)
			(* AppendToFile				DONE and TESTED DFB 20110602 *)
				(* Set CurrOperation	DONE and TESTED DFB 20110602 *)
				(* Busy, Done			DONE and TESTED DFB 20110602 *)
				(* Change state			DONE and TESTED DFB 20110602 *)
			(* Delete					DONE and TESTED DFB 20110602 *)
				(* Set CurrOperation	DONE and TESTED DFB 20110602 *)
				(* Busy, Done			DONE and TESTED DFB 20110602 *)
				(* Change state			DONE and TESTED DFB 20110602 *)
		(* Reset Done					DONE and TESTED DFB 20110602 *)

	(* ST_OPEN							DONE and TESTED DFB 20110602 *)
		(* FUB inputs					DONE and TESTED DFB 20120131 *)
		(* Status checking				DONE and TESTED DFB 20110602 *)
			(* Done						DONE and TESTED DFB 20110602 *)
			(* No error					DONE and TESTED DFB 20110602 *)
				(* Open					DONE and TESTED DFB 20110602 *)
				(* SaveAs				DONE and TESTED DFB 20110602 *)
				(* AppendToFile			DONE and TESTED DFB 20110602 *)
			(* File not found			DONE and TESTED DFB 20111222 *)
				(* Open					DONE and TESTED DFB 20111222 *)
				(* SaveAs				DONE and TESTED DFB 20111222 *)
				(* AppendToFile			DONE and TESTED DFB 20111222 *)
			(* Other error				DONE and TESTED DFB 20111222 *)

	(* ST_CREATE						DONE and TESTED DFB 20110602 *)
		(* FUB inputs					DONE and TESTED DFB 20120131 *)
		(* Status checking				DONE and TESTED DFB 20110602 *)
			(* Done						DONE and TESTED DFB 20110602 *)
			(* No error					DONE and TESTED DFB 20110602 *)
				(* SaveAs				DONE and TESTED DFB 20110602 *)
				(* AppendToFile			DONE and TESTED DFB 20110602 *)
			(* Error					DONE will not be tested *)

	(* ST_READ							DONE and TESTED DFB 20110602 *)
		(* FUB inputs					DONE and TESTED DFB 20120131 *)
		(* Status checking				DONE and TESTED DFB 20110602 *)
			(* Done						DONE and TESTED DFB 20110602 *)
			(* No error					DONE and TESTED DFB 20110602 *)
			(* Error					DONE and TESTED DFB 20111222 *)

	(* ST_WRITE							DONE and TESTED DFB 20110602 *)
		(* FUB inputs					DONE and TESTED DFB 20120131 *)
			(* SaveAs					DONE and TESTED DFB 20120131 *)
			(* AppendToFile				DONE and TESTED DFB 20120131 *)
				(* No error				DONE and TESTED DFB 20120131 *)
				(* MaxFileSize error	DONE and TESTED DFB 20120131 *)
		(* Status checking				DONE and TESTED DFB 20110602 *)
			(* Done						DONE and TESTED DFB 20110602 *)
			(* No error					DONE and TESTED DFB 20110602 *)
			(* Error					DONE and TESTED DFB 20111222 *)

	(* ST_CLOSE							DONE and TESTED DFB 20110602 *)
		(* FUB inputs					DONE and TESTED DFB 20120131 *)
		(* Status checking				DONE and TESTED DFB 20110602 *)
			(* Done						DONE and TESTED DFB 20110602 *)
			(* No error					DONE and TESTED DFB 20110602 *)
				(* ErrorClose			DONE and TESTED DFB 20110602 *)
			(* Error					DONE will not be tested *)

	(* ST_DELETE						DONE and TESTED DFB 20110602 *)
		(* FUB inputs					DONE and TESTED DFB 20120131 *)
		(* Status checking				DONE and TESTED DFB 20110602 *)
			(* Done						DONE and TESTED DFB 20110602 *)
			(* No error					DONE and TESTED DFB 20111222 *)
			(* File not found			DONE and TESTED DFB 20111222 *)
			(* Other error				DONE and TESTED DFB 20111222 *)

	(* ST_ERROR							DONE and TESTED DFB 20110602 *)
		(* Disable FUBs					DONE and TESTED DFB 20110602 *)
		(* AcknowledgeError CMD			DONE and TESTED DFB 20111222 *)

(* Busy, Done, Error					DONE and TESTED DFB 20111222 *)

FUNCTION FIOWrapFn_Cyclic

(************************************************************************)
(* Set return value to get rid of compiler warning 						*)
(************************************************************************)

	FIOWrapFn_Cyclic:=	FALSE;

	(************************************************************************)
	(* Reset internal CMDs													*)
	(************************************************************************)

	IF( NOT(t.IN.CMD.Open) )THEN

		t.Internal.CMD.Open:=	0;

	END_IF

	IF( NOT(t.IN.CMD.SaveAs) )THEN

		t.Internal.CMD.SaveAs:=	0;

	END_IF

	IF( NOT(t.IN.CMD.AppendToFile) )THEN

		t.Internal.CMD.AppendToFile:=	0;

	END_IF

	IF( NOT(t.IN.CMD.Delete) )THEN

		t.Internal.CMD.Delete:=	0;

	END_IF

	(************************************************************************)
	(* Main state machine													*)
	(************************************************************************)

	CASE t.Internal.State OF

		FIOWRAP_ST_WAIT:

			(* If all CMDs are cleared, then clear Done status *)

			IF( 	NOT(t.IN.CMD.Open)
				AND	NOT(t.IN.CMD.SaveAs)
				AND	NOT(t.IN.CMD.AppendToFile)
				AND	NOT(t.IN.CMD.Delete)
				)THEN

				t.OUT.STAT.Done:=	0;

			END_IF

			(* Set CurrOperation to INVALID. It will be set below on leaving the state *)

			t.Internal.CurrOperation:=	FIOWRAP_OP_INVALID;

			(* Wait for new commands *)

			IF( t.IN.CMD.SaveAs AND NOT(t.Internal.CMD.SaveAs) )THEN

				t.Internal.CMD.SaveAs:=	1;

				t.OUT.STAT.Busy:=	1;
				t.OUT.STAT.Done:=	0;

				t.Internal.State:=			FIOWRAP_ST_OPEN;
				t.Internal.CurrOperation:=	FIOWRAP_OP_SAVEAS;

			ELSIF( t.IN.CMD.Open AND NOT(t.Internal.CMD.Open) )THEN

				t.Internal.CMD.Open:=	1;

				t.OUT.STAT.Busy:=	1;
				t.OUT.STAT.Done:=	0;

				t.Internal.State:=			FIOWRAP_ST_OPEN;
				t.Internal.CurrOperation:=	FIOWRAP_OP_OPEN;

			ELSIF( t.IN.CMD.AppendToFile AND NOT(t.Internal.CMD.AppendToFile) )THEN

				t.Internal.CMD.AppendToFile:=	1;

				t.OUT.STAT.Busy:=	1;
				t.OUT.STAT.Done:=	0;

				t.Internal.State:=			FIOWRAP_ST_OPEN;
				t.Internal.CurrOperation:=	FIOWRAP_OP_APPEND;

			ELSIF( t.IN.CMD.Delete AND NOT(t.Internal.CMD.Delete) )THEN

				t.Internal.CMD.Delete:=	1;

				t.OUT.STAT.Busy:=	1;
				t.OUT.STAT.Done:=	0;

				t.Internal.State:=			FIOWRAP_ST_DELETE;
				t.Internal.CurrOperation:=	FIOWRAP_OP_INVALID;

			END_IF

			// Reset internal fileCreated whenever done goes false
			t.Internal.FileCreated := t.Internal.FileCreated AND t.OUT.STAT.Done;

		FIOWRAP_ST_OPEN:

			(* Open file *)

			t.Internal.FUB.Open.enable:=	1;
			t.Internal.FUB.Open.pDevice:=	ADR(t.IN.PAR.FileDevice);
			t.Internal.FUB.Open.pFile:=		ADR(t.IN.PAR.FileName);
			t.Internal.FUB.Open.mode:=		fiREAD_WRITE;

			(* Check status *)

			IF( t.Internal.FUB.Open.status < FIOWRAP_STAT_DISABLED ) THEN

				(* Turn off FUB *)

				t.Internal.FUB.Open.enable:=	0;

				IF( t.Internal.FUB.Open.status = FIOWRAP_STAT_OK ) THEN

				(* All good
					Get Ident, go to appropriate state *)

					t.Internal.FileID:=		t.Internal.FUB.Open.ident;
					t.Internal.FileLen:=	t.Internal.FUB.Open.filelen;

					IF( t.Internal.CurrOperation = FIOWRAP_OP_OPEN ) THEN

						t.Internal.State:=	FIOWRAP_ST_READ;

					ELSIF( 		(t.Internal.CurrOperation = FIOWRAP_OP_SAVEAS)
						OR	(t.Internal.CurrOperation = FIOWRAP_OP_APPEND)
						)THEN

						t.Internal.State:=	FIOWRAP_ST_WRITE;

					ELSE

						fiowSetError( DINT_TO_UINT(FIOWRAP_ERR_INVALIDOP), t );

					END_IF (* check for reading or writing *)

				ELSIF( t.Internal.FUB.Open.status = fiERR_FILE_NOT_FOUND ) THEN

				(* File not found
					If reading, error
					If writing, create file *)

					IF( t.Internal.CurrOperation = FIOWRAP_OP_OPEN ) THEN

						fiowSetError( t.Internal.FUB.Open.status, t );

					ELSIF( 		(t.Internal.CurrOperation = FIOWRAP_OP_SAVEAS)
						OR	(t.Internal.CurrOperation = FIOWRAP_OP_APPEND)
						)THEN

						t.Internal.State:=	FIOWRAP_ST_CREATE;

					ELSE

						fiowSetError( DINT_TO_UINT(FIOWRAP_ERR_INVALIDOP), t );

					END_IF (* Check for reading or writing *)

				ELSE

					(* Other error *)

					fiowSetError( t.Internal.FUB.Open.status, t );

				END_IF (* If error *)

			END_IF (* If done *)

		FIOWRAP_ST_CREATE:

			(* Create file *)

			t.Internal.FUB.Create.enable:=	1;
			t.Internal.FUB.Create.pDevice:=	ADR( t.IN.PAR.FileDevice );
			t.Internal.FUB.Create.pFile:=	ADR( t.IN.PAR.FileName );

			(* Check status *)

			IF( t.Internal.FUB.Create.status < FIOWRAP_STAT_DISABLED ) THEN

				(* Turn off FUB *)

				t.Internal.FUB.Create.enable:=	0;

				IF( t.Internal.FUB.Create.status = FIOWRAP_STAT_OK ) THEN

					(* All good, grab ident, go to write state *)

					t.Internal.FileID:=		t.Internal.FUB.Create.ident;
					t.Internal.FileLen:=	0;
					t.Internal.FileCreated:= 1;

					IF( 	(t.Internal.CurrOperation = FIOWRAP_OP_SAVEAS)
						OR	(t.Internal.CurrOperation = FIOWRAP_OP_APPEND)
						)THEN

						t.Internal.State:=	FIOWRAP_ST_WRITE_HEADER;

					ELSE

						fiowSetError( DINT_TO_UINT(FIOWRAP_ERR_INVALIDOP), t );

					END_IF (* Check for writing *)

				ELSE

					(* Error *)

					fiowSetError( t.Internal.FUB.Create.status, t );

				END_IF (* If error *)

			END_IF (* If done *)

		FIOWRAP_ST_WRITE_HEADER:

			// skip this if no header
			IF t.IN.PAR.pHeader = 0 OR t.IN.PAR.headerLen = 0 THEN

				t.Internal.State:=	FIOWRAP_ST_WRITE;

			ELSE

				t.Internal.FUB.Write.enable:=	1;
				t.Internal.FUB.Write.ident:=	t.Internal.FileID;

				t.Internal.FUB.Write.offset:=	0;

				t.Internal.FUB.Write.pSrc:=		t.IN.PAR.pHeader;
				t.Internal.headerLen:=			t.IN.PAR.headerLen;
				t.Internal.FUB.Write.len:=		t.Internal.headerLen;

				(* Check status *)

				IF( t.Internal.FUB.Write.status < FIOWRAP_STAT_DISABLED ) THEN

					(* Turn off FUB *)

					t.Internal.FUB.Write.enable:=	0;

					IF( t.Internal.FUB.Write.status = FIOWRAP_STAT_OK ) THEN

						t.Internal.FileLen:= t.IN.PAR.headerLen;
						(* All good, go to close state *)
						t.Internal.State:=	FIOWRAP_ST_WRITE;

					ELSE

						(* Error *)
						(* Since already opened file, need to close file before going to error state *)

						t.Internal.ErrorClose:=	1;

						fiowSetError( t.Internal.FUB.Write.status, t );

						t.Internal.State:=		FIOWRAP_ST_CLOSE;

					END_IF (* If error *)

				END_IF (* If done *)
			END_IF

		FIOWRAP_ST_READ:

			(* Read from file *)

			t.Internal.FUB.Read.enable:=	1;
			t.Internal.FUB.Read.ident:=		t.Internal.FileID;
			t.Internal.FUB.Read.offset:=	t.IN.PAR.offset;
			t.Internal.FUB.Read.pDest:=		t.IN.PAR.pData;
			t.Internal.FUB.Read.len:=		t.IN.PAR.len;

			(* Check status *)

			IF( t.Internal.FUB.Read.status < FIOWRAP_STAT_DISABLED ) THEN

				(* Turn off FUB *)

				t.Internal.FUB.Read.enable:=	0;

				IF( t.Internal.FUB.Read.status = FIOWRAP_STAT_OK ) THEN

					(* All good, go to close state *)

					t.Internal.State:=	FIOWRAP_ST_CLOSE;

				ELSE

					(* Error *)
					(* Since already opened file, need to close file before going to error state *)

					t.Internal.ErrorClose:=	1;

					fiowSetError( t.Internal.FUB.Read.status, t );

					t.Internal.State:=		FIOWRAP_ST_CLOSE;

				END_IF (* If error *)

			END_IF (* If done *)

		FIOWRAP_ST_WRITE:

			(* Write to file *)

			t.Internal.FUB.Write.enable:=	1;
			t.Internal.FUB.Write.ident:=	t.Internal.FileID;

			IF( t.Internal.CurrOperation = FIOWRAP_OP_SAVEAS )THEN

				// only offset write by header if the file is new
				IF t.Internal.FileCreated THEN
					t.Internal.FUB.Write.offset:= t.Internal.headerLen + t.IN.PAR.offset;
				ELSE
					t.Internal.FUB.Write.offset:=	t.IN.PAR.offset;
				END_IF

			ELSIF( 		(t.Internal.CurrOperation = FIOWRAP_OP_APPEND)
				AND	(t.Internal.FileLen + t.IN.PAR.len <= t.IN.PAR.MaxFileSize)
				)THEN

				t.Internal.FUB.Write.offset:=	t.Internal.FileLen;

			ELSIF( (t.Internal.CurrOperation = FIOWRAP_OP_APPEND)
				AND (t.IN.PAR.MultiFile)
				AND (t.Internal.FileLen <> 0)
				)THEN

				t.Internal.FUB.Write.enable:= 0;
				t.Internal.CurrOperation:= FIOWRAP_OP_APPEND_NEW;
				t.Internal.State:= FIOWRAP_ST_CLOSE;

			ELSE

				(* Error *)
				(* Since already opened file, need to close file before going to error state *)

				t.Internal.ErrorClose:=	1;
				t.Internal.FUB.Write.enable:=	0;

				fiowSetError( DINT_TO_UINT(FIOWRAP_ERR_MAXFILESIZE), t );

				t.Internal.State:=		FIOWRAP_ST_CLOSE;

			END_IF (* If error *)

			t.Internal.FUB.Write.pSrc:=		t.IN.PAR.pData;
			t.Internal.FUB.Write.len:=		t.IN.PAR.len;

			(* Check status *)

			IF( t.Internal.FUB.Write.status < FIOWRAP_STAT_DISABLED ) THEN

				(* Turn off FUB *)

				t.Internal.FUB.Write.enable:=	0;

				IF( t.Internal.FUB.Write.status = FIOWRAP_STAT_OK ) THEN

					(* All good, go to close state *)

					t.Internal.State:=	FIOWRAP_ST_CLOSE;

				ELSE

					(* Error *)
					(* Since already opened file, need to close file before going to error state *)

					t.Internal.ErrorClose:=	1;

					fiowSetError( t.Internal.FUB.Write.status, t );

					t.Internal.State:=		FIOWRAP_ST_CLOSE;

				END_IF (* If error *)

			END_IF (* If done *)

		FIOWRAP_ST_RENAME:

			t.Internal.FUB.Rename.enable := 1;

			(* Check status *)

			IF( t.Internal.FUB.Rename.status < FIOWRAP_STAT_DISABLED )THEN

				(* Turn off FUB *)

				t.Internal.FUB.Rename.enable:= 0;

				IF ( t.Internal.FUB.Rename.status = FIOWRAP_STAT_OK ) THEN

					IF( t.Internal.CurrOperation = FIOWRAP_OP_APPEND ) THEN

						t.Internal.State:= FIOWRAP_ST_OPEN;

					ELSE

						t.Internal.State:= FIOWRAP_ST_WAIT;

					END_IF

				ELSE

					(* Error *)

					fiowSetError( t.Internal.FUB.Rename.status, t );

				END_IF

			ELSIF( t.Internal.FUB.Rename.status = FIOWRAP_STAT_DISABLED )THEN

				(* Get file name and extension *)
				SplitFileName(ADR(t.IN.PAR.FileName), ADR(t.Internal.Name), ADR(t.Internal.Extension));

				IF (NOT (brsstrcmp(ADR(t.IN.PAR.Suffix), ADR('')) = 0)) THEN
					t.Internal.newFileName := CONCAT(t.Internal.Name, CONCAT(t.IN.PAR.Suffix, CONCAT('.', t.Internal.Extension)));

				ELSE
					(* Get Time *)
					t.Internal.FUB.GetTime.enable := TRUE;
					t.Internal.FUB.GetTime();

					IF( t.Internal.FUB.GetTime.status = 0 )THEN

						(* Generate Timestamp *)
						(* YYYY-MM-DD_HH-MM-SS *)
						//GenerateTimestamp(t.Internal.FUB.GetTime.DT1, ADR(t.Internal.Timestamp), SIZEOF(t.Internal.Timestamp));
						DT_TO_DTStructure( t.Internal.FUB.GetTime.DT1, ADR(t.Internal.DTStruct) );
						brsitoa(t.Internal.DTStruct.year, ADR(t.Internal.TempStr));
						t.Internal.Timestamp := CONCAT(t.Internal.TempStr,'-'); // Year
						brsitoa(t.Internal.DTStruct.month, ADR(t.Internal.TempStr));
						t.Internal.Timestamp := CONCAT(t.Internal.Timestamp, CONCAT(t.Internal.TempStr, '-')); // Month
						brsitoa(t.Internal.DTStruct.day, ADR(t.Internal.TempStr));
						t.Internal.Timestamp := CONCAT(t.Internal.Timestamp, CONCAT(t.Internal.TempStr, '_')); // Day
						brsitoa(t.Internal.DTStruct.hour, ADR(t.Internal.TempStr));
						t.Internal.Timestamp := CONCAT(t.Internal.Timestamp, CONCAT(t.Internal.TempStr, '-')); // Hour
						brsitoa(t.Internal.DTStruct.minute, ADR(t.Internal.TempStr));
						t.Internal.Timestamp := CONCAT(t.Internal.Timestamp, CONCAT(t.Internal.TempStr, '-')); // Min
						brsitoa(t.Internal.DTStruct.second, ADR(t.Internal.TempStr));
						t.Internal.Timestamp := CONCAT(t.Internal.Timestamp, t.Internal.TempStr); // Second

						(* Combine name with timestamp *)
						(* NAME_TIMESTAMP.EXTENSION *)
						t.Internal.newFileName := CONCAT(t.Internal.Name, CONCAT('_', CONCAT(t.Internal.Timestamp, CONCAT('.', t.Internal.Extension))));
						//t.Internal.newFileName := CONCAT(t.IN.PAR.FileName, t.Internal.Timestamp);
						//t.IN.PAR.FileName
					ELSE

						t.Internal.newFileName := CONCAT(t.Internal.Name, CONCAT('-old.', t.Internal.Extension));

					END_IF

				END_IF

				t.Internal.FUB.Rename.pDevice := ADR(t.IN.PAR.FileDevice);
				t.Internal.FUB.Rename.pName := ADR(t.IN.PAR.FileName);
				t.Internal.FUB.Rename.pNewName := ADR(t.Internal.newFileName);

			END_IF

		FIOWRAP_ST_CLOSE:

			(* Close file *)

			t.Internal.FUB.Close.enable:=	1;
			t.Internal.FUB.Close.ident:=	t.Internal.FileID;

			(* Check status *)

			IF( t.Internal.FUB.Close.status < FIOWRAP_STAT_DISABLED ) THEN

				(* Turn off FUB *)

				t.Internal.FUB.Close.enable:=	0;

				IF( t.Internal.FUB.Close.status = FIOWRAP_STAT_OK ) THEN

					IF( t.Internal.ErrorClose ) THEN

						(* If error close, go to error state *)

						t.Internal.State:=	FIOWRAP_ST_ERROR;

					ELSIF( t.Internal.CurrOperation = FIOWRAP_OP_APPEND_NEW )THEN

						(* continue with appending *)

						t.Internal.CurrOperation:= FIOWRAP_OP_APPEND;
						t.Internal.State:= FIOWRAP_ST_RENAME;
					ELSE

						(* otherwise, done, set status and go to wait state *)

						t.Internal.State:=	FIOWRAP_ST_INFO;

					END_IF (* If ErrorClose *)

				ELSE

					(* Error *)

					fiowSetError( t.Internal.FUB.Close.status, t );

				END_IF (* If error *)

			END_IF (*If done *)

		FIOWRAP_ST_DELETE:

			(* Delete file *)

			t.Internal.FUB.Delete.enable:=	1;
			t.Internal.FUB.Delete.pDevice:=	ADR(t.IN.PAR.FileDevice);
			t.Internal.FUB.Delete.pName:=	ADR(t.IN.PAR.FileName);

			(* Check status *)

			IF( t.Internal.FUB.Delete.status < FIOWRAP_STAT_DISABLED ) THEN

				(* Turn off FUB *)

				t.Internal.FUB.Delete.enable:=	0;

				IF( 	(t.Internal.FUB.Delete.status = FIOWRAP_STAT_OK)
					OR	(t.Internal.FUB.Delete.status = fiERR_FILE_NOT_FOUND)
					)THEN

					(* Done, set status and go to wait state *)

					t.OUT.STAT.Busy:=	0;
					t.OUT.STAT.Done:=	1;

					t.Internal.State:=	FIOWRAP_ST_WAIT;

				ELSE

					(* Error *)

					fiowSetError( t.Internal.FUB.Delete.status, t );

				END_IF (* If error *)

			END_IF (*If done *)

		FIOWRAP_ST_INFO:
			t.Internal.FUB.Info.enable := 1;
			t.Internal.FUB.Info.pDevice := ADR(t.IN.PAR.FileDevice);
			t.Internal.FUB.Info.pName := ADR(t.IN.PAR.FileName);
			t.Internal.FUB.Info.pInfo := ADR(t.Internal.FileInfo);

			(* Check status *)
			IF( t.Internal.FUB.Info.status < FIOWRAP_STAT_DISABLED ) THEN
				(* Turn off FUB *)
				t.Internal.FUB.Info.enable:=	0;
				IF(t.Internal.FUB.Info.status = FIOWRAP_STAT_OK)THEN
					t.Internal.FileLen := t.Internal.FileInfo.size;
					t.OUT.STAT.Busy:=	0;
					t.OUT.STAT.Done:=	1;
					t.Internal.State:=	FIOWRAP_ST_WAIT;
				ELSE
					(* Error *)
					fiowSetError( t.Internal.FUB.Info.status, t );
				END_IF (* If error *)
			END_IF (*If done *)

		FIOWRAP_ST_ERROR:

			(* Turn off all FUBs, just in case *)

			t.Internal.FUB.Open.enable:=	0;
			t.Internal.FUB.Create.enable:=	0;
			t.Internal.FUB.Read.enable:=	0;
			t.Internal.FUB.Write.enable:=	0;
			t.Internal.FUB.Close.enable:=	0;
			t.Internal.FUB.Delete.enable:=	0;
			t.Internal.FUB.Rename.enable:=	0;
			t.Internal.FUB.GetTime.enable:= 0;

			IF( t.IN.CMD.AcknowledgeError )THEN

				t.OUT.STAT.Error:=			0;
				t.OUT.STAT.ErrorID:=		0;
				t.OUT.STAT.ErrorString:=	'';
				t.OUT.STAT.ErrorLevel:=		0;
				t.Internal.ErrorClose:=		0;
				t.Internal.State:=			FIOWRAP_ST_WAIT;

			END_IF

	END_CASE

	// Copy curent file length to output
	t.OUT.STAT.FileLen := t.Internal.FileLen;

	(* Reset AcknowledgeError CMD *)

	t.IN.CMD.AcknowledgeError:=	0;

	(****************************************)
	(* Call FUBs							*)
	(****************************************)

	t.Internal.FUB.Open();
	t.Internal.FUB.Create();
	t.Internal.FUB.Read();
	t.Internal.FUB.Write();
	t.Internal.FUB.Close();
	t.Internal.FUB.Delete();
	t.Internal.FUB.Rename();
	t.Internal.FUB.Info();

	(****************************************)
	(* Set ReadyForCMD						*)
	(****************************************)

	t.OUT.STAT.NewFile:= t.Internal.FileCreated AND t.OUT.STAT.Done;
	t.OUT.STAT.ReadyForCMD:=		NOT(t.OUT.STAT.Busy)
	AND NOT(t.OUT.STAT.Done)
	AND	NOT(t.OUT.STAT.Error);

END_FUNCTION
